FUNCTION_BLOCK FB_ArrManip
VAR_INPUT
END_VAR
VAR_OUTPUT
END_VAR
VAR
END_VAR

METHOD flip
VAR_INPUT
	arr : REFERENCE TO ARRAY [1..NUMLEVELS] OF INT;
END_VAR
VAR
	i, mid : INT;
	bfr : INT;
END_VAR
mid := NUMLEVELS/2;
FOR i:=1 TO mid DO
	bfr := arr[i];
	arr[i] := arr[NUMLEVELS+1-i];
	arr[NUMLEVELS+1-i] := bfr;
END_FOR
END_METHOD

METHOD index : INT
VAR_INPUT
	arr : REFERENCE TO ARRAY [1..NUMLEVELS] OF BOOL;
END_VAR
VAR
	i : INT;
END_VAR
(* 
Method returns the index of the first element that is TRUE.
If all Elements are zero, the return value is 0.
*)

FOR i:=1 TO NUMLEVELS DO
	IF arr[i] = TRUE THEN
		index := i;
		RETURN;
	END_IF
END_FOR

index := 0;
END_METHOD

METHOD insert : BOOL
VAR_INPUT
	arr : REFERENCE TO ARRAY [1..NUMLEVELS] OF INT;
	newElement : INT;
	freeElement : INT;
END_VAR
VAR 
	i : INT;
END_VAR
FOR i:=1 TO NUMLEVELS DO
	IF arr[i] = newElement THEN
		insert := TRUE;
		RETURN;
	END_IF
END_FOR

FOR i:=1 TO NUMLEVELS DO
	IF arr[i] = freeElement THEN
		arr[i] := newElement;
		insert := TRUE;
		RETURN;
	END_IF
END_FOR

insert := FALSE;
END_METHOD

METHOD isElement : BOOL
VAR_INPUT
	arr : REFERENCE TO ARRAY [1..NUMLEVELS] OF INT;
	entry : INT;
END_VAR
VAR
	i : INT;
END_VAR
FOR i:=1 TO NUMLEVELS DO
	IF arr[i] = entry THEN
		isELement := TRUE;
		RETURN;
	END_IF
END_FOR
isElement := FALSE;
END_METHOD

METHOD isEmpty : BOOL
VAR_INPUT
	arr : REFERENCE TO ARRAY [1..NUMLEVELS] OF INT;
	emptyElement : INT;
END_VAR
VAR
	i : INT;
END_VAR
FOR i:=1 TO NUMLEVELS DO
	IF arr[i] <> emptyElement THEN
		isEmpty := FALSE;
		RETURN;
	END_IF
END_FOR
isEmpty := TRUE;
END_METHOD

METHOD PRIVATE partition : INT
VAR_INPUT
	arr : REFERENCE TO ARRAY [1..NUMLEVELS] OF INT;
	lo, hi : INT;
END_VAR
VAR
	pivot : INT;
	i, j : INT;
	bfr : INT;
END_VAR
pivot := arr[hi];
i := lo;

FOR j:=lo TO hi DO
	IF arr[j] < pivot THEN
		bfr := arr[i];
		arr[i] := arr[j];
		arr[j] := bfr;
		i := i+1;
	END_IF
END_FOR

bfr := arr[i];
arr[i] := arr[hi];
arr[hi] := bfr;

partition := i;
END_METHOD

METHOD pop_front : INT
VAR_INPUT
	arr : REFERENCE TO ARRAY [1..NUMLEVELS] OF INT;
	fill : INT;
END_VAR
VAR
	nOut : INT;
	i : INT;
END_VAR
nOut := arr[1];

FOR i:=1 TO NUMLEVELS-1 DO
	arr[i] := arr[i+1];
END_FOR
arr[NUMLEVELS] := fill;

pop_front := nOut;
END_METHOD

METHOD quicksort_asc
VAR_INPUT
	arr : REFERENCE TO ARRAY [1..NUMLEVELS] OF INT;
	lo, hi : INT;
END_VAR
VAR
	p : INT;
END_VAR
IF lo < hi THEN
	p := partition(arr, lo, hi);
	quicksort_asc(arr, lo, p-1);
	quicksort_asc(arr, p+1, hi);
END_IF
END_METHOD

METHOD quicksort_desc
VAR_INPUT
	arr : REFERENCE TO ARRAY [1..NUMLEVELS] OF INT;
	lo, hi : INT;
END_VAR
VAR
	p : INT;
END_VAR
quicksort_asc(arr:=arr, lo:=lo, hi:=hi);
flip(arr:=arr);
END_METHOD

END_FUNCTION_BLOCK

(* stored: Version 1.1.0.1, ProductVersion 3.1.4024.6
   POU FB_ArrManip: Id {3caf019d-58bd-4837-9068-c953846ad35b}, SpecialFunc None
   Method flip: Id {a15c0025-8bae-40c2-8706-69ea6e75a6dc}
   Method index: Id {5f9aef16-fcb2-419f-b21e-f2b69f686cab}
   Method insert: Id {915327af-0e91-41e0-be8c-81ad65b793fd}
   Method isElement: Id {cf569ec2-295d-4af6-9c82-730bcb265787}
   Method isEmpty: Id {09f2da74-234d-44c7-a057-7b449b4ef231}
   Method partition: Id {d0bc2153-5e93-40d1-8f10-f56185e95095}
   Method pop_front: Id {4e3c8a1b-db7e-40fa-aee8-9e3588f3917f}
   Method quicksort_asc: Id {8e7d33b3-d623-4bb0-8e47-176e7e919ed0}
   Method quicksort_desc: Id {7c8882d7-643c-4714-8ac1-90c814fe9bcb} *)
